FUNCTION TryConvert_LINT_TO_BOOL : BOOL
VAR_INPUT
	in : LINT;
	out : REFERENCE TO BOOL;
END_VAR

out := LINT_TO_BOOL(in);
TryConvert_LINT_TO_BOOL := TRUE;

END_FUNCTION

(* stored: Version 1.1.0.1, ProductVersion 3.1.4024.12
   POU TryConvert_LINT_TO_BOOL: Id {6e0ed1b7-ae64-4290-832e-b3cc95e27c7c}, SpecialFunc None *)
